(* PLC project MQTT, OpenPLC MQTT 1.0, author OpenPLC Lib Writter *)
(* stored: creationDateTime 2023-04-26T04:54:00, modificationDateTime 2023-04-26T04:54:00 *)

(* Receive MQTT messages for a particular TOPIC when RECEIVE is active. You must subscribe to a topic first before you can start receiving messages for that particular topic. Once a message is received, RECEIVED output is triggered, and MESSAGE will contain the received message as a STRING. *)
FUNCTION_BLOCK MQTT_RECEIVE
  VAR_INPUT
    RECEIVE : BOOL;  (* RECEIVE *)
    TOPIC : STRING;  (* TOPIC *)
  END_VAR
  VAR_OUTPUT
    RECEIVED : BOOL;  (* RECEIVED *)
    MESSAGE : STRING;  (* MESSAGE *)
  END_VAR

  RECEIVED := 0;
END_FUNCTION_BLOCK

(* Sends a MESSAGE to a particular TOPIC when SEND input is triggered. Keep in mind that SEND is not configured as a rising edge input, which means that MQTT_SEND will continuously send messages every scan cycle while SEND is TRUE. If the message was sent without errors, SUCCESS will be TRUE. *)
FUNCTION_BLOCK MQTT_SEND
  VAR_INPUT
    SEND : BOOL;  (* SEND *)
    TOPIC : STRING;  (* TOPIC *)
    MESSAGE : STRING;  (* MESSAGE *)
  END_VAR
  VAR_OUTPUT
    SUCCESS : BOOL;  (* SUCCESS *)
  END_VAR

  SUCCESS := 0;
END_FUNCTION_BLOCK

(* Connect to a BROKER at a given PORT when CONNECT is triggered. If a successfull connection is made, SUCCESS is set to TRUE *)
FUNCTION_BLOCK MQTT_CONNECT
  VAR_INPUT
    CONNECT : BOOL;  (* CONNECT *)
    BROKER : STRING;  (* BROKER *)
    PORT : UINT;  (* PORT *)
  END_VAR
  VAR_OUTPUT
    SUCCESS : BOOL;  (* SUCCESS *)
  END_VAR

  SUCCESS := 0;
END_FUNCTION_BLOCK

(* Connect to an authenticated BROKER at a given PORT using the credentials from USER and PASSWORD when CONNECT is triggered. If a successfull connection is made, SUCCESS is set to TRUE *)
FUNCTION_BLOCK MQTT_CONNECT_AUTH
  VAR_INPUT
    CONNECT : BOOL;  (* CONNECT *)
    BROKER : STRING;  (* BROKER *)
    PORT : UINT;  (* PORT *)
    USER : STRING;  (* USER *)
    PASSWORD : STRING;  (* PASSWORD *)
  END_VAR
  VAR_OUTPUT
    SUCCESS : BOOL;  (* SUCCESS *)
  END_VAR

  SUCCESS := 0;
END_FUNCTION_BLOCK

(* Subscribe to a given TOPIC when SUBSCRIBE input is triggered. Upon a successfull subscription, SUCCESS is set to TRUE. Keep in mind that once you subscribe to a topic, OpenPLC will start receiving messages sent to that topic and storing them in a message pool. You must use the MQTT_RECEIVE block to retrieve messages from the pool and free up space to receive more messages. The maximum pool size is currently limited to 10 messages. If you let messages accumulate in the pool you will start loosing messages once the pool is full. *)
FUNCTION_BLOCK MQTT_SUBSCRIBE
  VAR_INPUT
    SUBSCRIBE : BOOL;  (* SUBSCRIBE *)
    TOPIC : STRING;  (* TOPIC *)
  END_VAR
  VAR_OUTPUT
    SUCCESS : BOOL;  (* SUCCESS *)
  END_VAR

  SUCCESS := 0;
END_FUNCTION_BLOCK

(* Unsubscribe to a given TOPIC when UNSUBSCRIBE input is triggered. Upon a successfull unsubscription, SUCCESS is set to TRUE. Keep in mind that once you unsubscribe to a topic, OpenPLC will stop storing messages sent to that topic in the message pool. However, messages received previously and not captured with a MQTT_RECEIVE block will remain in the pool using up pool space. *)
FUNCTION_BLOCK MQTT_UNSUBSCRIBE
  VAR_INPUT
    UNSUBSCRIBE : BOOL;  (* UNSUBSCRIBE *)
    TOPIC : STRING;  (* TOPIC *)
  END_VAR
  VAR_OUTPUT
    SUCCESS : BOOL;  (* SUCCESS *)
  END_VAR

  SUCCESS := 0;
END_FUNCTION_BLOCK

(* Disconnects from the current broker when DISCONNECT is set to TRUE. Upon a successfull disconnection, SUCCESS is set to TRUE. *)
FUNCTION_BLOCK MQTT_DISCONNECT
  VAR_INPUT
    DISCONNECT : BOOL;  (* DISCONNECT *)
  END_VAR
  VAR_OUTPUT
    SUCCESS : BOOL;  (* SUCCESS *)
  END_VAR

  SUCCESS := 0;
END_FUNCTION_BLOCK
